PROGRAM MAIN
VAR
	// Italian Pizza Margherita (via declaration)
	fbItalianStyle				: FB_PizzaItalianStyle;
	fbTomato					: FB_DecoratorTomato(fbItalianStyle, TRUE);
	fbCheese					: FB_DecoratorCheese(fbTomato);
	ipPizza						: I_Pizza := fbCheese;
	
	// Italian Pizza Margherita (via runtime)
	(* fbItalianStyle			: FB_PizzaItalianStyle;
	fbTomato					: FB_DecoratorTomato(0, FALSE);
	fbCheese					: FB_DecoratorCheese(0);
	ipPizza						: I_Pizza; *)
	
	bCreate						: BOOL;
	fPrice						: LREAL;
	sDescription				: STRING;
END_VAR

(* IF (bCreate) THEN
	bCreate := FALSE;
	fbTomato.ipDecorator := fbItalianStyle;
	fbCheese.ipDecorator := fbTomato;
	ipPizza := fbCheese;
END_IF *)

IF (ipPizza <> 0) THEN
	fPrice := ipPizza.GetPrice();
	sDescription := ipPizza.GetDescription();
END_IF

END_PROGRAM

(* stored: Version 1.1.0.1, ProductVersion 3.1.4022.16
   POU MAIN: Id {c9752a19-1ec4-4b65-9b03-7aba295e5266}, SpecialFunc None *)
